FUNCTION_BLOCK FB_Dog EXTENDS FB_Animal

VAR
	 y : INT:=76;
END_VAR

x := 876;

METHOD M_Bark
VAR_INPUT
END_VAR
THIS^.sOutput := 'Dog barks';
END_METHOD

END_FUNCTION_BLOCK

(* stored: Version 1.1.0.1, ProductVersion 3.1.4024.16
   POU FB_Dog: Id {2eaeca28-b8d7-4f4d-94d7-10072515f52f}, SpecialFunc None
   Method M_Bark: Id {f1496114-ddb4-46b1-ae38-84cb2ec324b4} *)
